// TwinCAT 3 PLC project Publisher
// ProgramVersion: 3.1.4022.0
// libraries:
//   Tc2_Standard, * (Beckhoff Automation GmbH)
//   Tc2_System, * (Beckhoff Automation GmbH)
//   Tc3_EventLogger, * (Beckhoff Automation GmbH)
//   Tc3_Module, * (Beckhoff Automation GmbH)
// project tree:
//   POUs/ E_Subsystem.TcDUT, FB_LogMessage.TcPOU, MAIN.TcPOU
//   / PublisherTask.TcTTO
// real-time tasks:
//   TASK PublisherTask: cycle T#10ms, priority 20, ADS port 350
//   TASK ListenerTask: cycle T#10ms, priority 1, ADS port 351

CONFIGURATION Publisher
    RESOURCE PLC ON TwinCAT3
        TASK PublisherTask(INTERVAL := T#10ms, PRIORITY := 20);
        PROGRAM MAIN WITH PublisherTask : MAIN;
    END_RESOURCE
END_CONFIGURATION

// ---- POUs/E_Subsystem.TcDUT
//LCLS Defined subsystems, make sure these correspond with casSubsystems in FB_LogMessage
TYPE E_Subsystem :
(
	UNKNOWN := 0, //Undefined system
	VACUUM := 1, //Vacuum control system
	MPS := 2, //Machine protection system
	MOTION := 3, //Motion control systems
	FIELDBUS := 4, //EtherCAT networks
	SDS := 5 //Sample delivery system
)WORD;
END_TYPE

// ---- POUs/MAIN.TcPOU
PROGRAM MAIN
VAR
	nSendMessage : UINT;
	bRaiseAlarm : BOOL;
	bConfirmAlarm : BOOL;
	bClearAlarm: BOOL;

	fbLogger : FB_TcEventLogger;
	fbMessage : FB_TcMessage;
	fbAlarm : FB_TcAlarm;
	bIsInitalized : BOOL;
	
	bSetJsonAttribute : BOOL;
	sJsonAttribute : STRING := '{"key":"value"}';
	
	msg : FB_LogMessage;
	hr : HRESULT;
	hrLastError : HRESULT;
	iCycle: INT;
END_VAR

iCycle := iCycle + 1;

IF (iCycle MOD 1000) = 0 THEN
	msg(sMsg:='cycle 1k', eSevr:=TcEventSeverity.Error);
END_IF
 
IF NOT bIsInitalized THEN
	bIsInitalized := TRUE;
	hr := fbAlarm.CreateEx(TC_EVENTS.PublisherEventClass.Alarm, TRUE, 0);
	IF FAILED(hr) THEN
		hrLastError := hr;
	END_IF
	//hr := fbMessage.CreateEx(TC_EVENTS.PublisherEventClass.Message, 0);
	hr := fbMessage.CreateEx(TC_EVENTS.TcGeneralAdsEventClass.Aborted, 0);
	IF FAILED(hr) THEN
		hrLastError := hr;
	END_IF
END_IF

IF bSetJsonAttribute THEN
	bSetJsonAttribute := FALSE;
	hr := fbAlarm.SetJsonAttribute(sJsonAttribute);
	IF FAILED(hr) THEN
		hrLastError := hr;
	END_IF
	hr := fbMessage.SetJsonAttribute(sJsonAttribute);
	IF FAILED(hr) THEN
		hrLastError := hr;
	END_IF
END_IF

WHILE nSendMessage > 0 DO
	hr := fbMessage.Send(0);
	IF FAILED(hr) THEN
		hrLastError := hr;
	END_IF
	nSendMessage := nSendMessage - 1;
END_WHILE

IF bRaiseAlarm THEN
	bRaiseAlarm := FALSE;
	hr := fbAlarm.Raise(0);
	IF FAILED(hr) THEN
		hrLastError := hr;
	END_IF
END_IF

IF bConfirmAlarm THEN
	bConfirmAlarm := FALSE;
	hr := fbAlarm.Confirm(0);
	IF FAILED(hr) THEN
		hrLastError := hr;
	END_IF
END_IF

IF bClearAlarm THEN
	bClearAlarm := FALSE;
	hr := fbAlarm.Clear(0, FALSE);
	IF FAILED(hr) THEN
		hrLastError := hr;
	END_IF
END_IF

END_PROGRAM

// ---- POUs/FB_LogMessage.TcPOU
{attribute 'reflection'}
FUNCTION_BLOCK FB_LogMessage
VAR_INPUT
	sMsg			: T_MaxString; 		// Message to send
	eSevr			: TcEventSeverity	:= TcEventSeverity.Verbose;
	eSubsystem		: E_Subsystem; 		// Subsystem TODO
	Json			: T_MaxString;		// JSON to add to the message
END_VAR

VAR_OUTPUT
END_VAR

VAR
	bInitialized		:	BOOL := FALSE;
	bInitFailed			:	BOOL := FALSE;
	sMessage 			:	T_MaxString;
	sSubsystemSource	:	STRING;
	fbMessage			:	REFERENCE TO FB_TcMessage;
	fbMessages 			:	ARRAY [1..5] OF FB_TcMessage;
	fbSource 			:	FB_TcSourceInfo;
	ipResultMessage	 	:	I_TcMessage;
	hr 					:	HRESULT;
	hrLastInternalError :	HRESULT;
	eTraceLevel 		:	TcEventSeverity := TcEventSeverity.Verbose;
	eEventEntry 		:	TcEventEntry;
	
	{attribute 'instance-path'} 
    {attribute 'noinit'} 
	sPath				:	T_MaxString;
END_VAR

IF NOT bInitialized AND NOT bInitFailed THEN
	hr := fbMessages[TC_EVENTS.LCLSLoggingEvent.Verbose.nEventId].CreateEx(TC_EVENTS.LCLSLoggingEvent.Verbose, 0 (*fbSource*) );
	IF FAILED(hr) THEN
		bInitFailed := TRUE;
		hrLastInternalError := hr;
	END_IF

	hr := fbMessages[TC_EVENTS.LCLSLoggingEvent.Warning.nEventId].CreateEx(TC_EVENTS.LCLSLoggingEvent.Warning, 0 (*fbSource*) );
	IF FAILED(hr) THEN
		bInitFailed := TRUE;
		hrLastInternalError := hr;
	END_IF

	hr := fbMessages[TC_EVENTS.LCLSLoggingEvent.Info.nEventId].CreateEx(TC_EVENTS.LCLSLoggingEvent.Info, 0 (*fbSource*) );
	IF FAILED(hr) THEN
		bInitFailed := TRUE;
		hrLastInternalError := hr;
	END_IF

	hr := fbMessages[TC_EVENTS.LCLSLoggingEvent.Error.nEventId].CreateEx(TC_EVENTS.LCLSLoggingEvent.Error, 0 (*fbSource*) );
	IF FAILED(hr) THEN
		bInitFailed := TRUE;
		hrLastInternalError := hr;
	END_IF

	hr := fbMessages[TC_EVENTS.LCLSLoggingEvent.Critical.nEventId].CreateEx(TC_EVENTS.LCLSLoggingEvent.Critical, 0 (*fbSource*) );
	IF FAILED(hr) THEN
		bInitFailed := TRUE;
		hrLastInternalError := hr;
	END_IF
	
	IF bInitFailed THEN
		ADSLOGSTR(
			msgCtrlMask := ADSLOG_MSGTYPE_ERROR, 
			msgFmtStr   := '[LOGGER] Initialization failed in %s', 
			strArg      := sPath,
		); 
	ELSE
		bInitialized := TRUE;
	END_IF
END_IF

IF bInitFailed THEN
	RETURN;
END_IF
	
// Map the message severity to the LCLSLoggingEvent:
CASE eSevr OF
	TcEventSeverity.Verbose: 	fbMessage REF= fbMessages[TC_EVENTS.LCLSLoggingEvent.Verbose.nEventId];
	TcEventSeverity.Warning:	fbMessage REF= fbMessages[TC_EVENTS.LCLSLoggingEvent.Warning.nEventId];
	TcEventSeverity.Info:		fbMessage REF= fbMessages[TC_EVENTS.LCLSLoggingEvent.Info.nEventId];		
	TcEventSeverity.Error:		fbMessage REF= fbMessages[TC_EVENTS.LCLSLoggingEvent.Error.nEventId]; 
	TcEventSeverity.Critical:	fbMessage REF= fbMessages[TC_EVENTS.LCLSLoggingEvent.Critical.nEventId];
	ELSE
		RETURN;
END_CASE

CASE eSubsystem OF
	E_Subsystem.FIELDBUS: 	sSubsystemSource := '/Fieldbus';
	E_Subsystem.MOTION: 	sSubsystemSource := '/Motion';
	E_Subsystem.MPS: 		sSubsystemSource := '/MPS';
	E_Subsystem.SDS: 		sSubsystemSource := '/SDS';
	E_Subsystem.VACUUM:		sSubsystemSource := '/Vacuum';	
	ELSE
		sSubsystemSource := '/Unknown';
END_CASE

// Clearing the source here will clear the event GUID, causing the message to not be resolved.
// However, we can change the name as desired:
//fbSource.Clear();
fbSource.sName := CONCAT(sPath, sSubsystemSource);

ipResultMessage := fbMessage;
hr := fbMessage.CreateEx(stEventEntry:=ipResultMessage.stEventEntry, ipSourceInfo:=fbSource);

// This is where the message text gets appended:
fbMessage.ipArguments.Clear();
fbMessage.ipArguments.AddString(sMsg);

// For a final format of:
// 'Path.to.FB_LogMessage/Subsystem': {Unknown,Error,Warning,Verbose} (message)

IF NOT FAILED(hr) AND fbMessage.eSeverity >= eTraceLevel THEN
	hr := fbMessage.Send(0);
END_IF

IF FAILED(hr) THEN
	hrLastInternalError := hr;
END_IF

END_FUNCTION_BLOCK
